(* IEC 61131-3 sources: CodesysTest/export/Unused/FB_SimBasicVacuum.pou/VacuumOn.prop, 1 file *)

(* ---- Get.pm.st ---- *)
(*#-#-#-#-#-#-#-#-#-#---Declaration---#-#-#-#-#-#-#-#-#-#-#-#-#*)

VAR
END_VAR
(*#-#-#-#-#-#-#-#-#-#---Implementation---#-#-#-#-#-#-#-#-#-#-#-#-#*)

VacuumOn := startVac.Q;
